TYPE ST_APP_CTRL :
STRUCT
  Cmd       : E_INSTANCE_CMD;
  Variant   : E_APP_VARIANT;
END_STRUCT
END_TYPE

(* stored: Version 1.1.0.1
   DUT ST_APP_CTRL: Id {a6664517-aaf7-4d6f-b90c-256468254a32} *)
